INTERFACE I_MotionInterlocks

// this comes from I_MotionDriveShareData or could be provided by iMotionAxisCommon MC_Power Status block for non sync operation
PROPERTY Enable : BOOL
GET
END_GET
SET
END_SET
END_PROPERTY

PROPERTY Error : BOOL
GET
END_GET
END_PROPERTY

PROPERTY ErrorID : UDINT
GET
END_GET
END_PROPERTY

PROPERTY ErrorMessage : STRING
GET
END_GET
END_PROPERTY

PROPERTY LimHit : BOOL
GET
END_GET
END_PROPERTY

PROPERTY LimHitIdling : BOOL
GET
END_GET
END_PROPERTY

PROPERTY LimHitMoving : BOOL
GET
END_GET
END_PROPERTY

END_INTERFACE

(* stored: Version 1.1.0.1
   Itf I_MotionInterlocks: Id {7ac89254-d732-4980-b014-871a72f21fa7}
   Property Enable: Id {b3c0e406-7678-4a5f-be3f-af744a5aeff8}
   Get Get: Id {83665a33-f3ff-4b48-a011-25c120a8a2b2}
   Set Set: Id {12ffdc1b-0be2-42d3-9e30-6b1b1af017b6}
   Property Error: Id {e7bf6778-c6b9-4c5a-b105-4d2a2c94dadc}
   Get Get: Id {e4d10e81-4cda-4fea-b6c9-9cbe365e367c}
   Property ErrorID: Id {052a5e61-bd0b-473b-8c73-0685a48edd45}
   Get Get: Id {f9a6101a-75a4-46b6-a241-3924343635ff}
   Property ErrorMessage: Id {bf7b81d5-c154-46fb-b50d-9188e5c9721a}
   Get Get: Id {904bcd85-b16b-4196-9319-f47b5feeb0d9}
   Property LimHit: Id {00f31b83-20b0-4e18-bb57-b84a58adcd1b}
   Get Get: Id {dc48a399-6ef3-4f49-9589-4858181b8029}
   Property LimHitIdling: Id {a9898372-986c-4ee4-bc98-43640fd003f2}
   Get Get: Id {d9233391-3505-4407-ade5-ca790ab05516}
   Property LimHitMoving: Id {12768a8b-8e2d-462d-ac59-05ed276cdf42}
   Get Get: Id {f40fa498-6562-48ff-8455-7f34f6bbcf01} *)
